FUNCTION_BLOCK Manual_Left
VAR_INPUT
	Input1:BOOL;
	ManualCotrolSpeed	:	REAL;
END_VAR
VAR_OUTPUT
	Flag1:BOOL;
END_VAR
VAR
	temp1:MC_MoveVelocity;
	AxisStop:MC_Stop;
	trig1: F_TRIG;
END_VAR

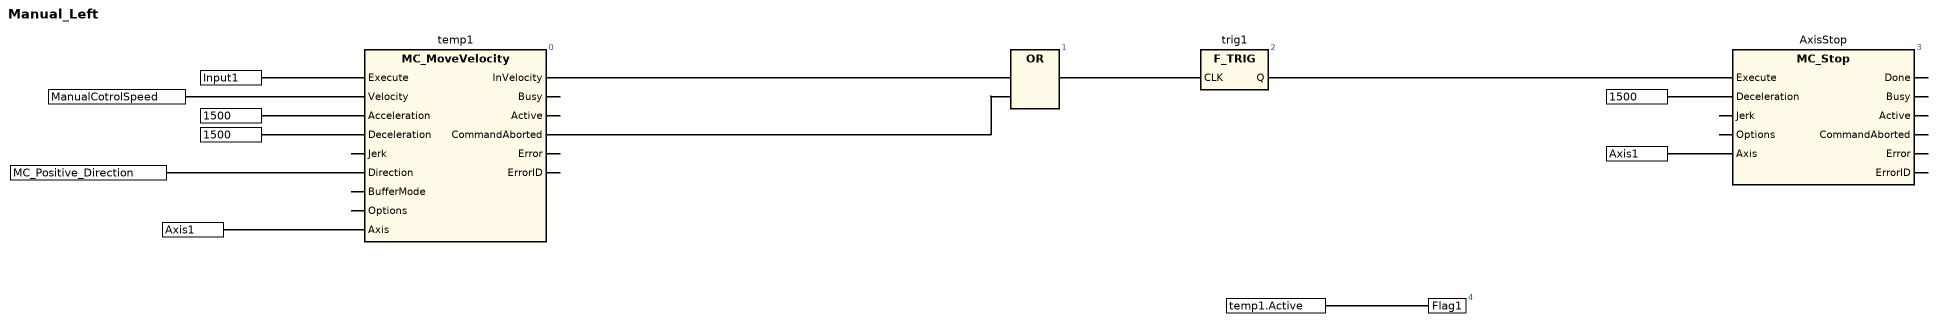
temp1(
    Execute := Input1,
    Velocity := ManualCotrolSpeed,
    Acceleration := 1500,
    Deceleration := 1500,
    Direction := MC_Positive_Direction,
    Axis := Axis1); // MC_MoveVelocity
trig1(CLK := temp1.InVelocity OR temp1.CommandAborted); // F_TRIG
AxisStop(Execute := trig1.Q, Deceleration := 1500, Axis := Axis1); // MC_Stop
Flag1 := temp1.Active;

END_FUNCTION_BLOCK

(* stored: Version 1.1.0.1, ProductVersion 3.1.4024.12
   POU Manual_Left: Id {d7e645b5-bc2e-4aa1-a68b-ad1c8595078c}, SpecialFunc None *)
